{attribute addProperty BoxType "EJ1957-0000-0017"}
{attribute addProperty Id "FSoE_CommandUSINT811FSOUT_Module_Module_FaultBIT10.1251FSIN_Module_1_Channel_1_InputBIT10.1251FSIN_Module_1_Channel_2_InputBIT10.1252FSIN_Module_1_Module_FaultBIT10.1251FSIN_Module_2_Channel_1_InputBIT10.1251FSIN_Module_2_Channel_2_InputBIT10.1252FSIN_Module_2_Module_FaultBIT10.1251FSIN_Module_3_Channel_1_InputBIT10.1251FSIN_Module_3_Channel_2_InputBIT10.1252FSIN_Module_3_Module_FaultBIT10.1251FSIN_Module_4_Channel_1_InputBIT10.1251FSIN_Module_4_Channel_2_InputBIT10.1252FSIN_Module_4_Module_FaultBIT10.1251FSoE_CRC_000UINT1623FSoE_Connection_IDUINT1622"}
{attribute addProperty CRC "139732654"}
{attribute addProperty SizeInBites "56"}
{attribute addProperty SizeInBytes "7"}
TYPE FSOE_085426AE :
STRUCT
	{attribute addProperty Name "FSoE_Command"}
	FSoE_Command : USINT;
	{attribute addProperty Name "FSOUT_Module_Module_Fault"}
	FSOUT_Module_Module_Fault : BOOL;
	{attribute addProperty Name "FSIN_Module_1_Channel_1_Input"}
	FSIN_Module_1_Channel_1_Input : BOOL;
	{attribute addProperty Name "FSIN_Module_1_Channel_2_Input"}
	FSIN_Module_1_Channel_2_Input : BOOL;
	{attribute addProperty Name "FSIN_Module_1_Module_Fault"}
	FSIN_Module_1_Module_Fault : BOOL;
	{attribute addProperty Name "FSIN_Module_2_Channel_1_Input"}
	FSIN_Module_2_Channel_1_Input : BOOL;
	{attribute addProperty Name "FSIN_Module_2_Channel_2_Input"}
	FSIN_Module_2_Channel_2_Input : BOOL;
	{attribute addProperty Name "FSIN_Module_2_Module_Fault"}
	FSIN_Module_2_Module_Fault : BOOL;
	{attribute addProperty Name "FSIN_Module_3_Channel_1_Input"}
	FSIN_Module_3_Channel_1_Input : BOOL;
	{attribute addProperty Name "FSIN_Module_3_Channel_2_Input"}
	FSIN_Module_3_Channel_2_Input : BOOL;
	{attribute addProperty Name "FSIN_Module_3_Module_Fault"}
	FSIN_Module_3_Module_Fault : BOOL;
	{attribute addProperty Name "FSIN_Module_4_Channel_1_Input"}
	FSIN_Module_4_Channel_1_Input : BOOL;
	{attribute addProperty Name "FSIN_Module_4_Channel_2_Input"}
	FSIN_Module_4_Channel_2_Input : BOOL;
	{attribute addProperty Name "FSIN_Module_4_Module_Fault"}
	FSIN_Module_4_Module_Fault : BOOL;
	{attribute 'hide'}
	reserve_1_BIT_0 : BOOL;
	{attribute 'hide'}
	reserve_1_BIT_1 : BOOL;
	{attribute 'hide'}
	reserve_1_BIT_2 : BOOL;
	{attribute addProperty Name "FSoE_CRC_000"}
	FSoE_CRC_000 : UINT;
	{attribute addProperty Name "FSoE_Connection_ID"}
	FSoE_Connection_ID : UINT;
END_STRUCT
END_TYPE

(* stored: Version 1.2.0.0, ProductVersion 3.1.4024.9
   DUT FSOE_085426AE: Id {b6ea8318-235d-45c1-b9d0-e8b60da585d0} *)
